SUBAPPLICATION GreenWhiteBackground_Auseinanderklappen (* Subapplication Type *)
  (* Standard: 61499-2 *)
  (* Version 1.0, 2023-02-11, franz *)
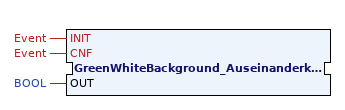
  EVENT_INPUT
    INIT;
    CNF;
  END_EVENT
  VAR_INPUT
    OUT : BOOL;
  END_VAR
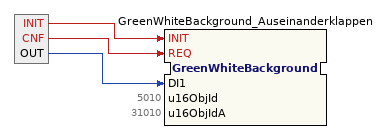
  FBS
    GreenWhiteBackground_Auseinanderklappen : GreenWhiteBackground(u16ObjId := 5010, u16ObjIdA := 31010);
  END_FBS
  EVENT_CONNECTIONS
    INIT TO GreenWhiteBackground_Auseinanderklappen.INIT;
    CNF TO GreenWhiteBackground_Auseinanderklappen.REQ;
  END_CONNECTIONS
  DATA_CONNECTIONS
    OUT TO GreenWhiteBackground_Auseinanderklappen.DI1;
  END_CONNECTIONS
END_SUBAPPLICATION
